TYPE "Positioning_DOL_Machine_DataIn"
VERSION : 0.1
// Block: Positioning_DOL_Machine_DataIn
   STRUCT
      PB : Ax_PB;
      LS_Minus : Bool;
      LS_Plus : Bool;
      Fan_M_ThermalProtection : Bool;
      Fan_M_Feedback : Bool;
      Brake_M_Q : Bool;
      Brake_M_Feedback : Bool;
   END_STRUCT;

END_TYPE
